(* Logix 5000 project; controller R5_CSS vendor 1 type 14 code 74 rev 19.11; software revision 19.01; part 6 of 20 *)
(* tags used below, declared in another part *)
   AC102A : ANALYTICAL;   // QUENCH WATER CONDUCTIVITY CONTROL
   FC101 : FLOW_CONTROL;   // QUENCH BASIN FLOW TRANSMITTER CONTROL
   FC108 : FLOW_CONTROL;   // QUENCH FEED FLOW TRANSMITTER
   FC140A : FLOW_CONTROL;   // QUENCH TOWER UPPER SPRAY FLOW CONTROL
   FC140B : FLOW_CONTROL;   // QUENCH TOWER LOWER SPRAY FLOW CONTROL
   FC215 : FLOW_CONTROL;   // OVERHEAD CONDENSER CHILLED WATER FLOW CONTROL
   FC365 : FLOW_CONTROL;   // COALESCER PROCESS IMPURITY FLOW CONTROL
   FC370 : FLOW_CONTROL;   // COALESCER MAKE UP WATER FLOW CONTROL
   FC403 : FLOW_CONTROL;   // COALESCER FLOW CONTROLLER FEEDS TCV108
   LCV370_Start : BOOL;
   PID_LC370_Enable : BOOL;
   TMR_FAULT : DINT;
(* MainProgram, continued *)

ROUTINE AT102A_QuenchWaterConductivity   (* ladder *)
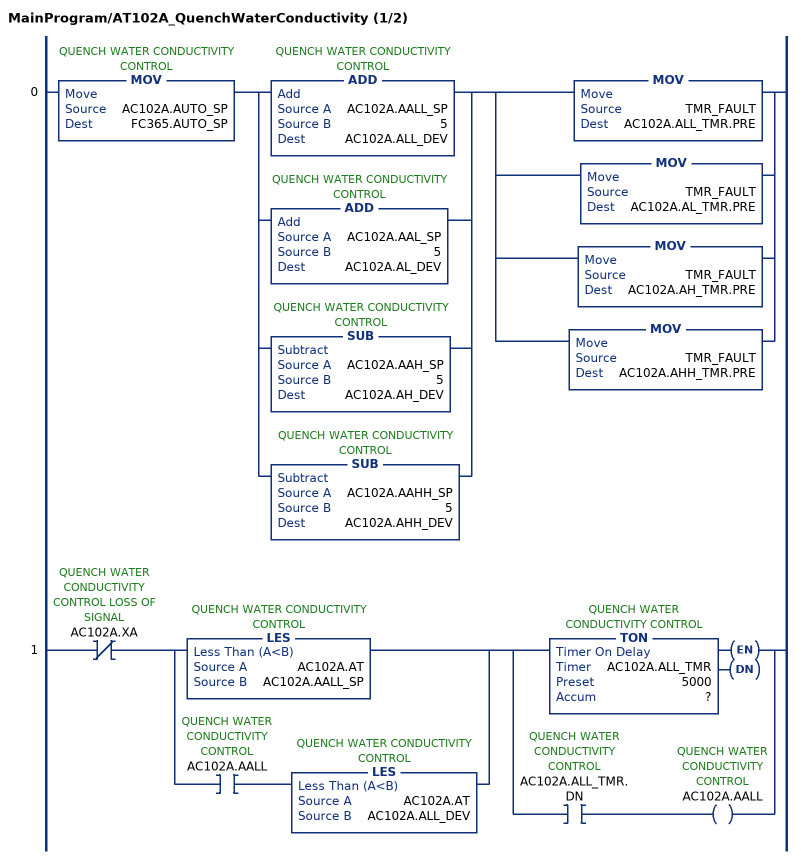
   0: MOV(AC102A.AUTO_SP,FC365.AUTO_SP)[ADD(AC102A.AALL_SP,5,AC102A.ALL_DEV) ,ADD(AC102A.AAL_SP,5,AC102A.AL_DEV) ,SUB(AC102A.AAH_SP,5,AC102A.AH_DEV) ,SUB(AC102A.AAHH_SP,5,AC102A.AHH_DEV) ][MOV(TMR_FAULT,AC102A.ALL_TMR.PRE) ,MOV(TMR_FAULT,AC102A.AL_TMR.PRE) ,MOV(TMR_FAULT,AC102A.AH_TMR.PRE) ,MOV(TMR_FAULT,AC102A.AHH_TMR.PRE) ];
   1: XIO(AC102A.XA)[LES(AC102A.AT,AC102A.AALL_SP) ,XIC(AC102A.AALL) LES(AC102A.AT,AC102A.ALL_DEV) ][TON(AC102A.ALL_TMR,?,?) ,XIC(AC102A.ALL_TMR.DN) OTE(AC102A.AALL) ];
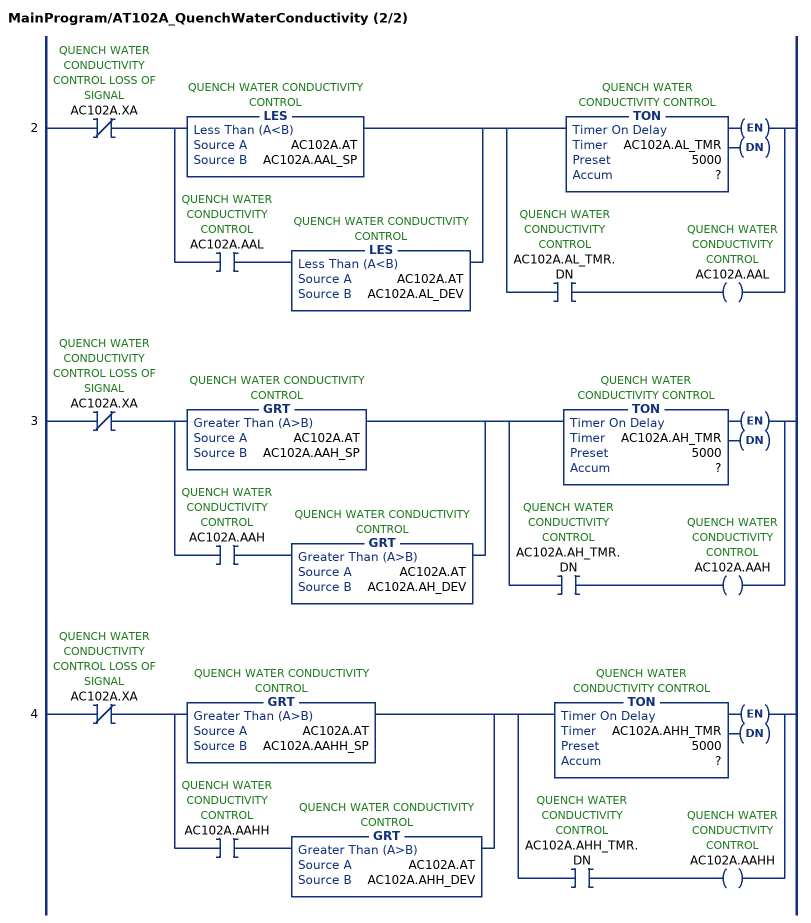
   2: XIO(AC102A.XA)[LES(AC102A.AT,AC102A.AAL_SP) ,XIC(AC102A.AAL) LES(AC102A.AT,AC102A.AL_DEV) ][TON(AC102A.AL_TMR,?,?) ,XIC(AC102A.AL_TMR.DN) OTE(AC102A.AAL) ];
   3: XIO(AC102A.XA)[GRT(AC102A.AT,AC102A.AAH_SP) ,XIC(AC102A.AAH) GRT(AC102A.AT,AC102A.AH_DEV) ][TON(AC102A.AH_TMR,?,?) ,XIC(AC102A.AH_TMR.DN) OTE(AC102A.AAH) ];
   4: XIO(AC102A.XA)[GRT(AC102A.AT,AC102A.AAHH_SP) ,XIC(AC102A.AAHH) GRT(AC102A.AT,AC102A.AHH_DEV) ][TON(AC102A.AHH_TMR,?,?) ,XIC(AC102A.AHH_TMR.DN) OTE(AC102A.AAHH) ];
END_ROUTINE

ROUTINE FC101_BasinFlow   (* ladder *)
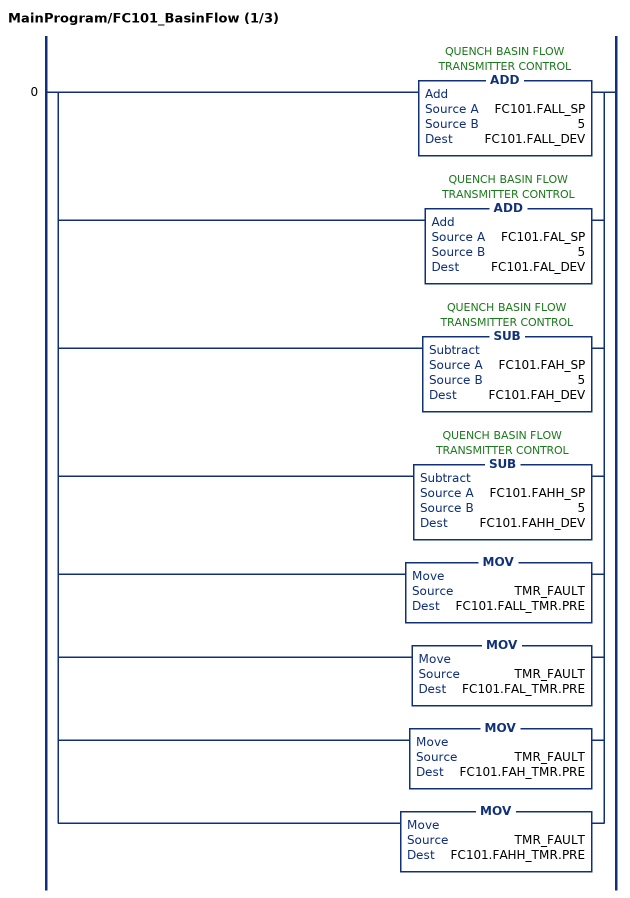
   0: [ADD(FC101.FALL_SP,5,FC101.FALL_DEV) ,ADD(FC101.FAL_SP,5,FC101.FAL_DEV) ,SUB(FC101.FAH_SP,5,FC101.FAH_DEV) ,SUB(FC101.FAHH_SP,5,FC101.FAHH_DEV) ,MOV(TMR_FAULT,FC101.FALL_TMR.PRE) ,MOV(TMR_FAULT,FC101.FAL_TMR.PRE) ,MOV(TMR_FAULT,FC101.FAH_TMR.PRE) ,MOV(TMR_FAULT,FC101.FAHH_TMR.PRE) ];
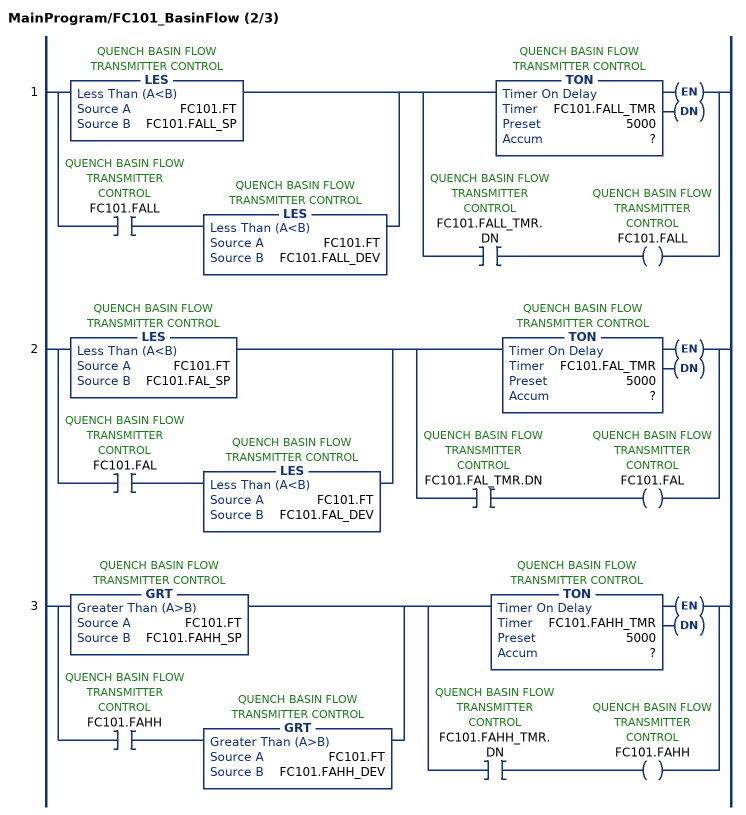
   1: [LES(FC101.FT,FC101.FALL_SP) ,XIC(FC101.FALL) LES(FC101.FT,FC101.FALL_DEV) ][TON(FC101.FALL_TMR,?,?) ,XIC(FC101.FALL_TMR.DN) OTE(FC101.FALL) ];
   2: [LES(FC101.FT,FC101.FAL_SP) ,XIC(FC101.FAL) LES(FC101.FT,FC101.FAL_DEV) ][TON(FC101.FAL_TMR,?,?) ,XIC(FC101.FAL_TMR.DN) OTE(FC101.FAL) ];
   3: [GRT(FC101.FT,FC101.FAHH_SP) ,XIC(FC101.FAHH) GRT(FC101.FT,FC101.FAHH_DEV) ][TON(FC101.FAHH_TMR,?,?) ,XIC(FC101.FAHH_TMR.DN) OTE(FC101.FAHH) ];
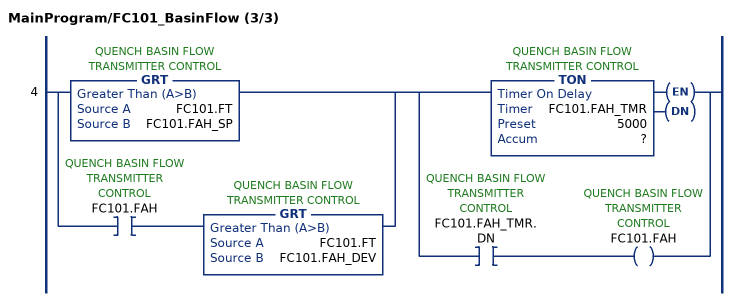
   4: [GRT(FC101.FT,FC101.FAH_SP) ,XIC(FC101.FAH) GRT(FC101.FT,FC101.FAH_DEV) ][TON(FC101.FAH_TMR,?,?) ,XIC(FC101.FAH_TMR.DN) OTE(FC101.FAH) ];
END_ROUTINE

ROUTINE FC108_QuenchTowerFlow   (* ladder *)
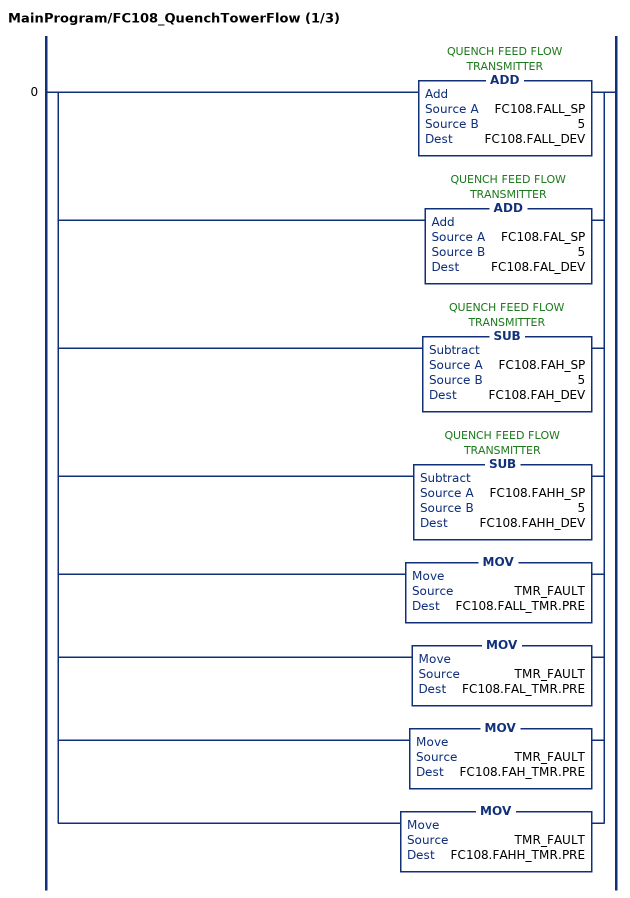
   0: [ADD(FC108.FALL_SP,5,FC108.FALL_DEV) ,ADD(FC108.FAL_SP,5,FC108.FAL_DEV) ,SUB(FC108.FAH_SP,5,FC108.FAH_DEV) ,SUB(FC108.FAHH_SP,5,FC108.FAHH_DEV) ,MOV(TMR_FAULT,FC108.FALL_TMR.PRE) ,MOV(TMR_FAULT,FC108.FAL_TMR.PRE) ,MOV(TMR_FAULT,FC108.FAH_TMR.PRE) ,MOV(TMR_FAULT,FC108.FAHH_TMR.PRE) ];
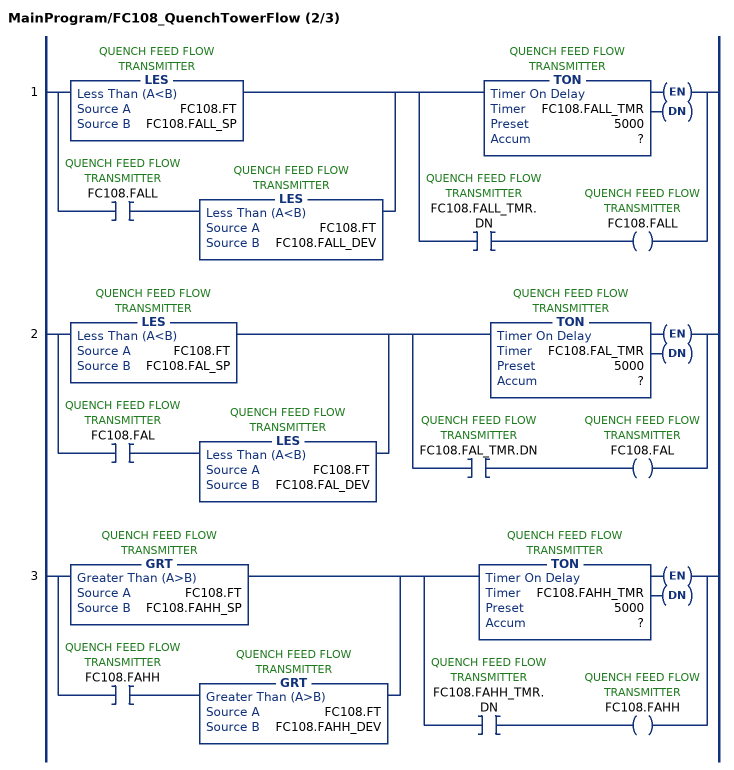
   1: [LES(FC108.FT,FC108.FALL_SP) ,XIC(FC108.FALL) LES(FC108.FT,FC108.FALL_DEV) ][TON(FC108.FALL_TMR,?,?) ,XIC(FC108.FALL_TMR.DN) OTE(FC108.FALL) ];
   2: [LES(FC108.FT,FC108.FAL_SP) ,XIC(FC108.FAL) LES(FC108.FT,FC108.FAL_DEV) ][TON(FC108.FAL_TMR,?,?) ,XIC(FC108.FAL_TMR.DN) OTE(FC108.FAL) ];
   3: [GRT(FC108.FT,FC108.FAHH_SP) ,XIC(FC108.FAHH) GRT(FC108.FT,FC108.FAHH_DEV) ][TON(FC108.FAHH_TMR,?,?) ,XIC(FC108.FAHH_TMR.DN) OTE(FC108.FAHH) ];
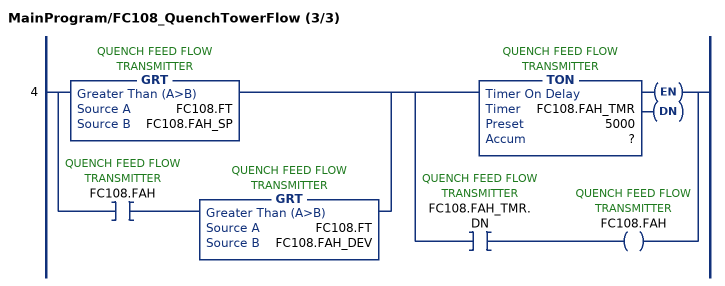
   4: [GRT(FC108.FT,FC108.FAH_SP) ,XIC(FC108.FAH) GRT(FC108.FT,FC108.FAH_DEV) ][TON(FC108.FAH_TMR,?,?) ,XIC(FC108.FAH_TMR.DN) OTE(FC108.FAH) ];
END_ROUTINE

ROUTINE FC140A_QuenchWaterUpperSprayFlow   (* ladder *)
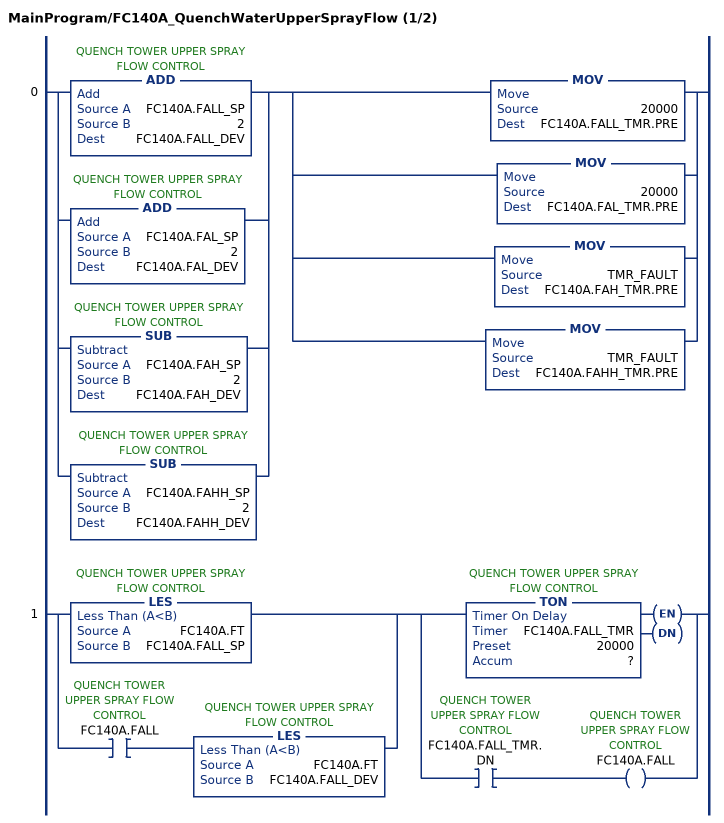
   0: [ADD(FC140A.FALL_SP,2,FC140A.FALL_DEV) ,ADD(FC140A.FAL_SP,2,FC140A.FAL_DEV) ,SUB(FC140A.FAH_SP,2,FC140A.FAH_DEV) ,SUB(FC140A.FAHH_SP,2,FC140A.FAHH_DEV) ][MOV(20000,FC140A.FALL_TMR.PRE) ,MOV(20000,FC140A.FAL_TMR.PRE) ,MOV(TMR_FAULT,FC140A.FAH_TMR.PRE) ,MOV(TMR_FAULT,FC140A.FAHH_TMR.PRE) ];
   1: [LES(FC140A.FT,FC140A.FALL_SP) ,XIC(FC140A.FALL) LES(FC140A.FT,FC140A.FALL_DEV) ][TON(FC140A.FALL_TMR,?,?) ,XIC(FC140A.FALL_TMR.DN) OTE(FC140A.FALL) ];
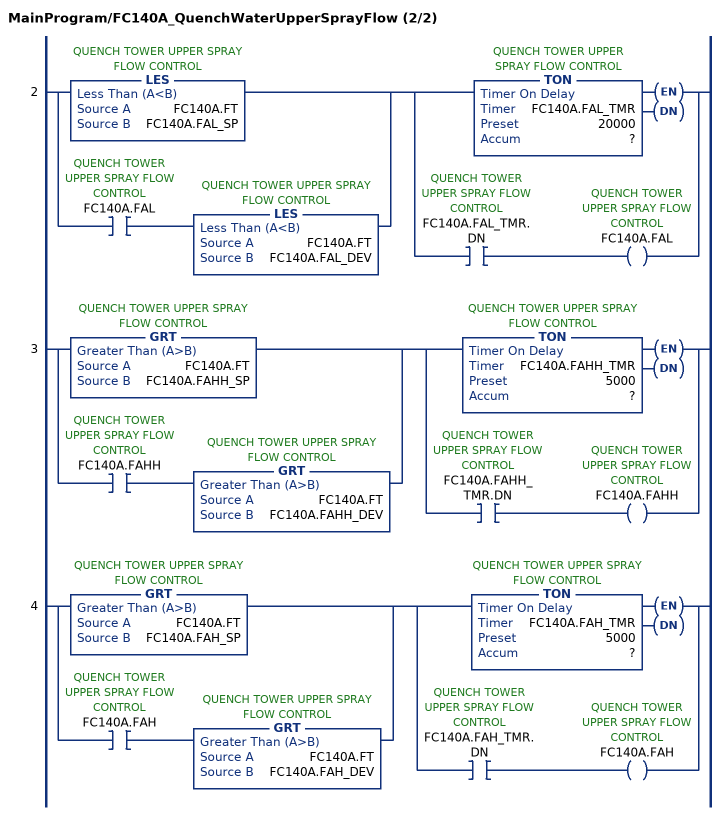
   2: [LES(FC140A.FT,FC140A.FAL_SP) ,XIC(FC140A.FAL) LES(FC140A.FT,FC140A.FAL_DEV) ][TON(FC140A.FAL_TMR,?,?) ,XIC(FC140A.FAL_TMR.DN) OTE(FC140A.FAL) ];
   3: [GRT(FC140A.FT,FC140A.FAHH_SP) ,XIC(FC140A.FAHH) GRT(FC140A.FT,FC140A.FAHH_DEV) ][TON(FC140A.FAHH_TMR,?,?) ,XIC(FC140A.FAHH_TMR.DN) OTE(FC140A.FAHH) ];
   4: [GRT(FC140A.FT,FC140A.FAH_SP) ,XIC(FC140A.FAH) GRT(FC140A.FT,FC140A.FAH_DEV) ][TON(FC140A.FAH_TMR,?,?) ,XIC(FC140A.FAH_TMR.DN) OTE(FC140A.FAH) ];
END_ROUTINE

ROUTINE FC140B_QuenchWaterLowerSprayFlow   (* ladder *)
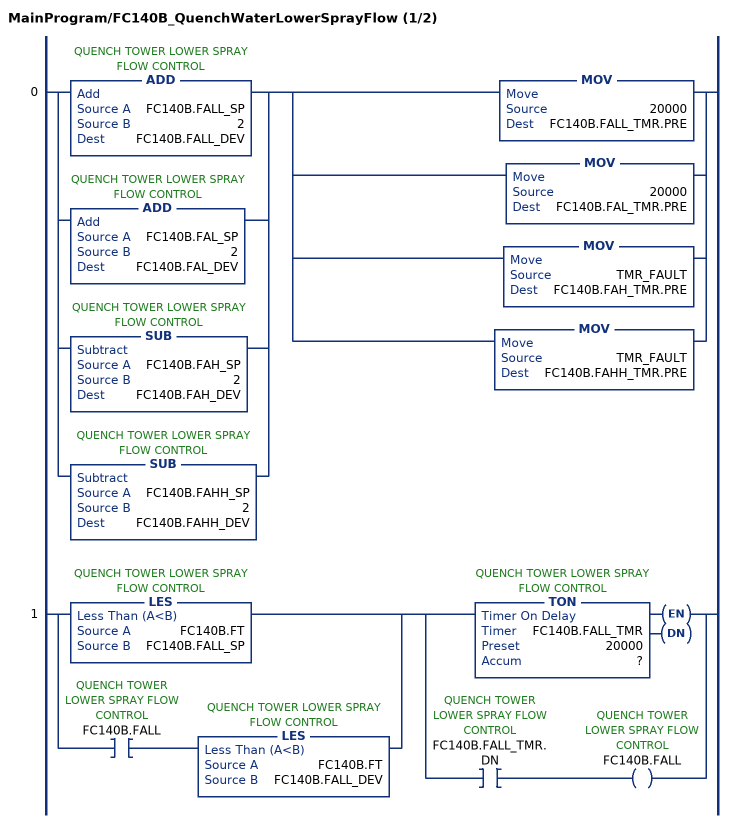
   0: [ADD(FC140B.FALL_SP,2,FC140B.FALL_DEV) ,ADD(FC140B.FAL_SP,2,FC140B.FAL_DEV) ,SUB(FC140B.FAH_SP,2,FC140B.FAH_DEV) ,SUB(FC140B.FAHH_SP,2,FC140B.FAHH_DEV) ][MOV(20000,FC140B.FALL_TMR.PRE) ,MOV(20000,FC140B.FAL_TMR.PRE) ,MOV(TMR_FAULT,FC140B.FAH_TMR.PRE) ,MOV(TMR_FAULT,FC140B.FAHH_TMR.PRE) ];
   1: [LES(FC140B.FT,FC140B.FALL_SP) ,XIC(FC140B.FALL) LES(FC140B.FT,FC140B.FALL_DEV) ][TON(FC140B.FALL_TMR,?,?) ,XIC(FC140B.FALL_TMR.DN) OTE(FC140B.FALL) ];
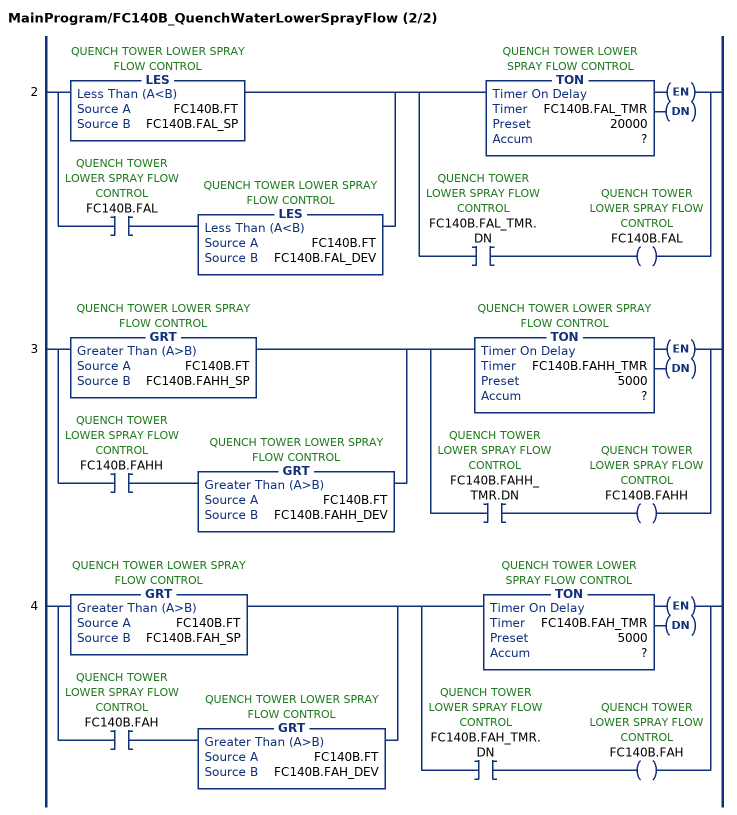
   2: [LES(FC140B.FT,FC140B.FAL_SP) ,XIC(FC140B.FAL) LES(FC140B.FT,FC140B.FAL_DEV) ][TON(FC140B.FAL_TMR,?,?) ,XIC(FC140B.FAL_TMR.DN) OTE(FC140B.FAL) ];
   3: [GRT(FC140B.FT,FC140B.FAHH_SP) ,XIC(FC140B.FAHH) GRT(FC140B.FT,FC140B.FAHH_DEV) ][TON(FC140B.FAHH_TMR,?,?) ,XIC(FC140B.FAHH_TMR.DN) OTE(FC140B.FAHH) ];
   4: [GRT(FC140B.FT,FC140B.FAH_SP) ,XIC(FC140B.FAH) GRT(FC140B.FT,FC140B.FAH_DEV) ][TON(FC140B.FAH_TMR,?,?) ,XIC(FC140B.FAH_TMR.DN) OTE(FC140B.FAH) ];
END_ROUTINE

ROUTINE FC215_OverheadCondChillWaterFlow   (* ladder *)
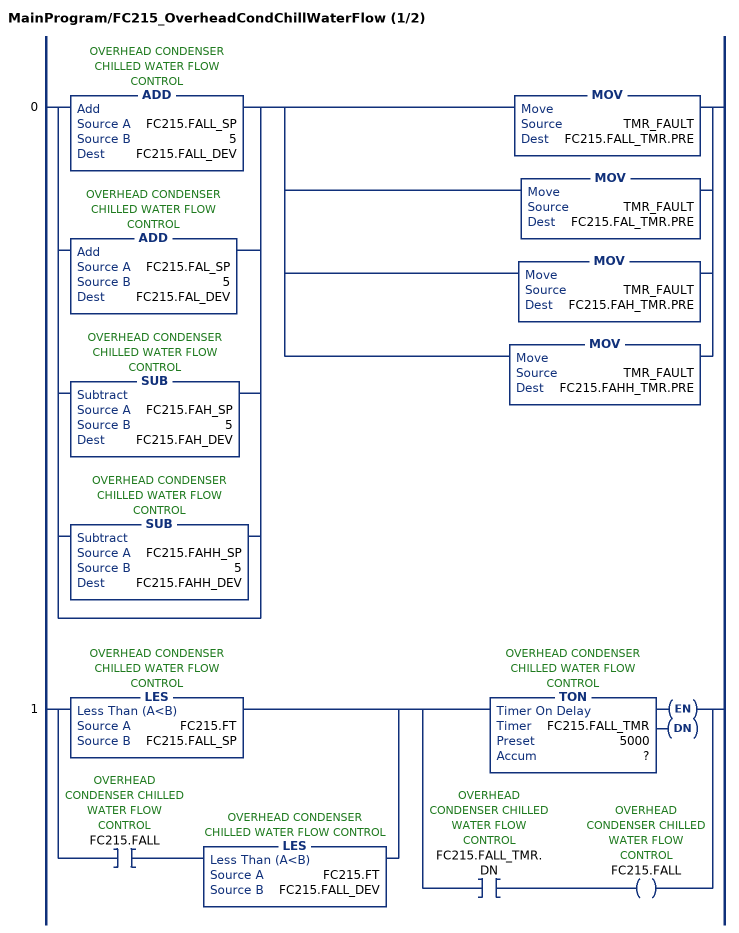
   0: [ADD(FC215.FALL_SP,5,FC215.FALL_DEV) ,ADD(FC215.FAL_SP,5,FC215.FAL_DEV) ,SUB(FC215.FAH_SP,5,FC215.FAH_DEV) ,SUB(FC215.FAHH_SP,5,FC215.FAHH_DEV) ,][MOV(TMR_FAULT,FC215.FALL_TMR.PRE) ,MOV(TMR_FAULT,FC215.FAL_TMR.PRE) ,MOV(TMR_FAULT,FC215.FAH_TMR.PRE) ,MOV(TMR_FAULT,FC215.FAHH_TMR.PRE) ];
   1: [LES(FC215.FT,FC215.FALL_SP) ,XIC(FC215.FALL) LES(FC215.FT,FC215.FALL_DEV) ][TON(FC215.FALL_TMR,?,?) ,XIC(FC215.FALL_TMR.DN) OTE(FC215.FALL) ];
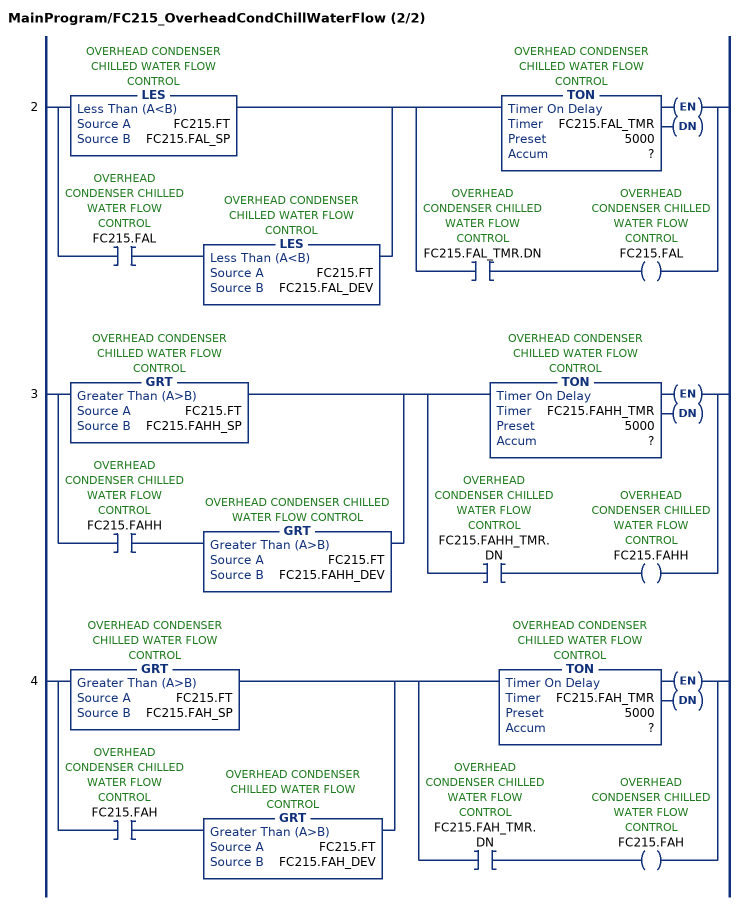
   2: [LES(FC215.FT,FC215.FAL_SP) ,XIC(FC215.FAL) LES(FC215.FT,FC215.FAL_DEV) ][TON(FC215.FAL_TMR,?,?) ,XIC(FC215.FAL_TMR.DN) OTE(FC215.FAL) ];
   3: [GRT(FC215.FT,FC215.FAHH_SP) ,XIC(FC215.FAHH) GRT(FC215.FT,FC215.FAHH_DEV) ][TON(FC215.FAHH_TMR,?,?) ,XIC(FC215.FAHH_TMR.DN) OTE(FC215.FAHH) ];
   4: [GRT(FC215.FT,FC215.FAH_SP) ,XIC(FC215.FAH) GRT(FC215.FT,FC215.FAH_DEV) ][TON(FC215.FAH_TMR,?,?) ,XIC(FC215.FAH_TMR.DN) OTE(FC215.FAH) ];
END_ROUTINE

ROUTINE FC370_WaterMakeupFlow   (* ladder *)
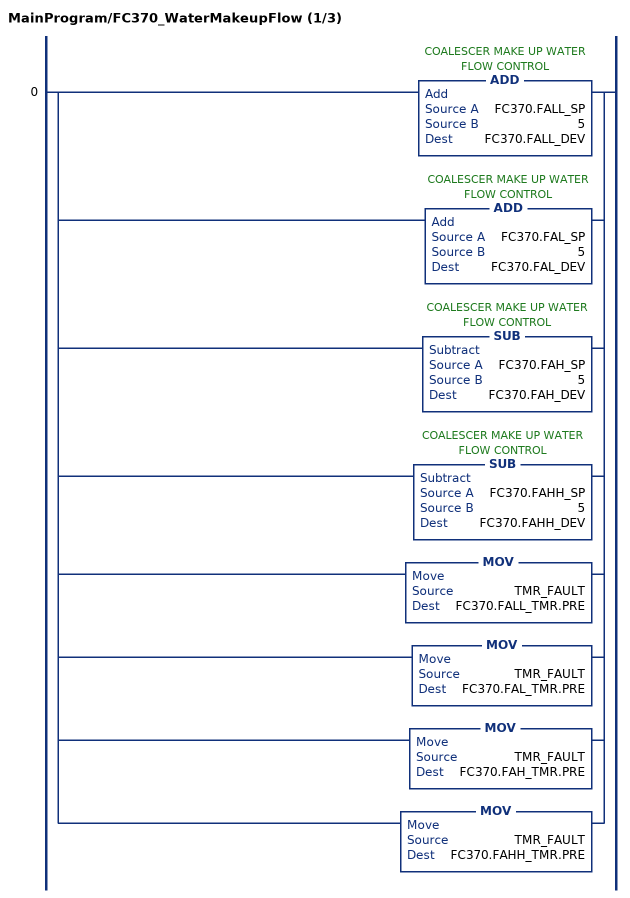
   0: [ADD(FC370.FALL_SP,5,FC370.FALL_DEV) ,ADD(FC370.FAL_SP,5,FC370.FAL_DEV) ,SUB(FC370.FAH_SP,5,FC370.FAH_DEV) ,SUB(FC370.FAHH_SP,5,FC370.FAHH_DEV) ,MOV(TMR_FAULT,FC370.FALL_TMR.PRE) ,MOV(TMR_FAULT,FC370.FAL_TMR.PRE) ,MOV(TMR_FAULT,FC370.FAH_TMR.PRE) ,MOV(TMR_FAULT,FC370.FAHH_TMR.PRE) ];
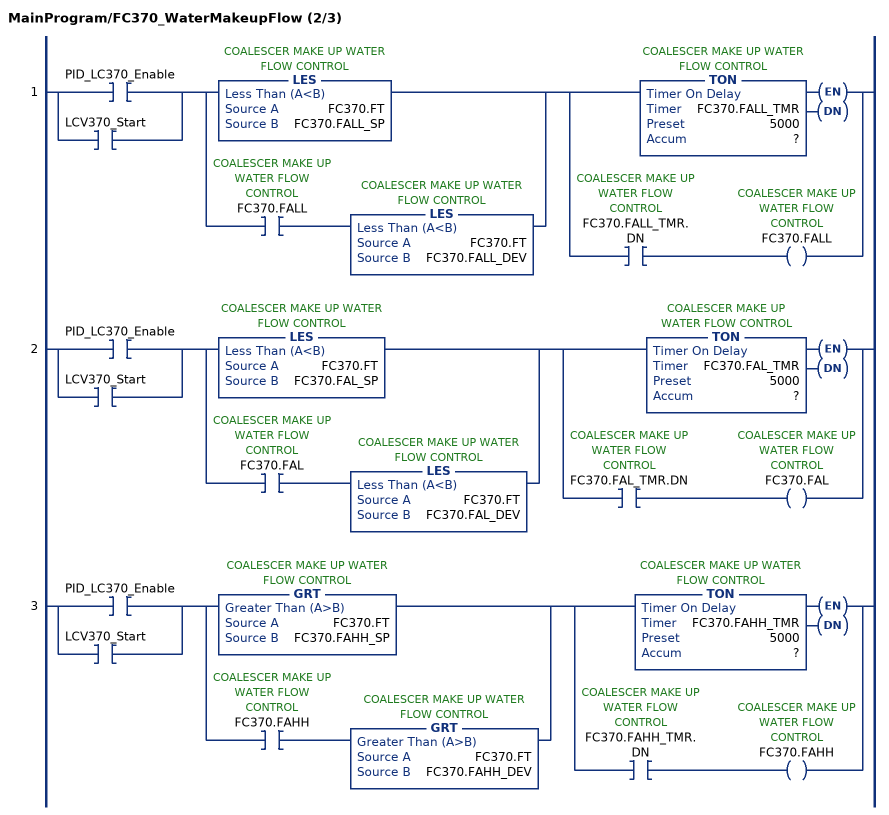
   1: [XIC(PID_LC370_Enable) ,XIC(LCV370_Start) ][LES(FC370.FT,FC370.FALL_SP) ,XIC(FC370.FALL) LES(FC370.FT,FC370.FALL_DEV) ][TON(FC370.FALL_TMR,?,?) ,XIC(FC370.FALL_TMR.DN) OTE(FC370.FALL) ];
   2: [XIC(PID_LC370_Enable) ,XIC(LCV370_Start) ][LES(FC370.FT,FC370.FAL_SP) ,XIC(FC370.FAL) LES(FC370.FT,FC370.FAL_DEV) ][TON(FC370.FAL_TMR,?,?) ,XIC(FC370.FAL_TMR.DN) OTE(FC370.FAL) ];
   3: [XIC(PID_LC370_Enable) ,XIC(LCV370_Start) ][GRT(FC370.FT,FC370.FAHH_SP) ,XIC(FC370.FAHH) GRT(FC370.FT,FC370.FAHH_DEV) ][TON(FC370.FAHH_TMR,?,?) ,XIC(FC370.FAHH_TMR.DN) OTE(FC370.FAHH) ];
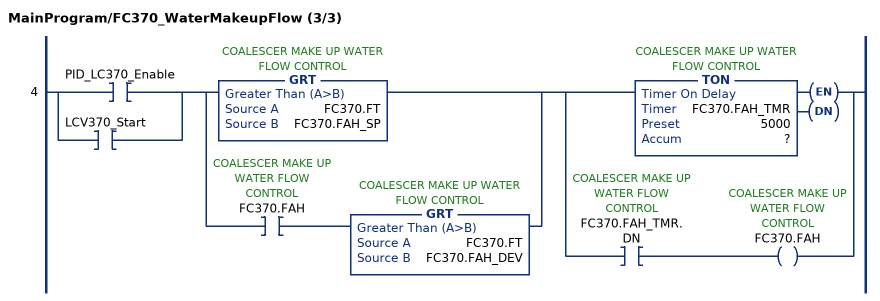
   4: [XIC(PID_LC370_Enable) ,XIC(LCV370_Start) ][GRT(FC370.FT,FC370.FAH_SP) ,XIC(FC370.FAH) GRT(FC370.FT,FC370.FAH_DEV) ][TON(FC370.FAH_TMR,?,?) ,XIC(FC370.FAH_TMR.DN) OTE(FC370.FAH) ];
END_ROUTINE

ROUTINE FC403_QuenchWaterTotalFlow   (* ladder *)
// COALESCER FLOW CONTROL
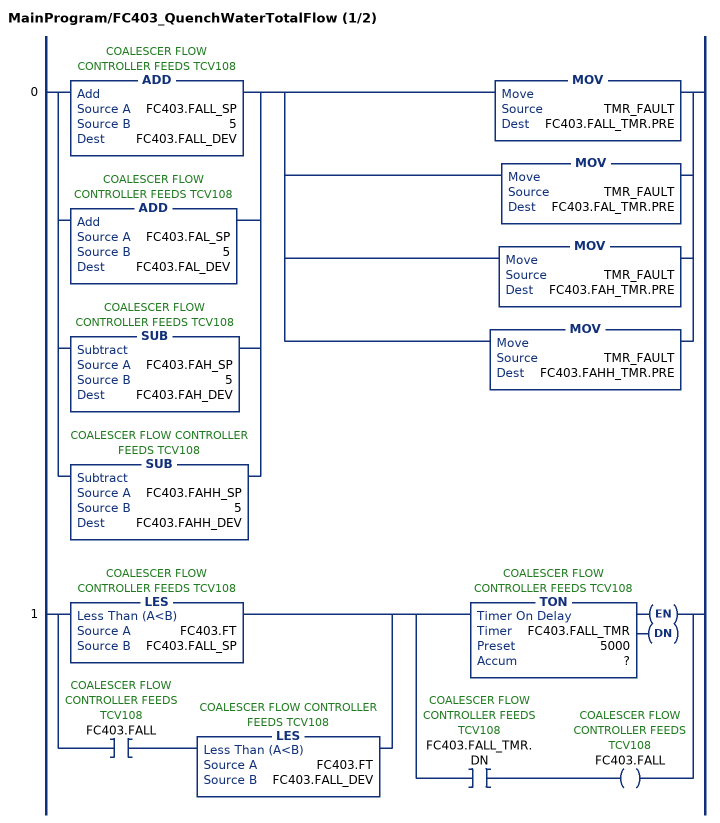
   0: [ADD(FC403.FALL_SP,5,FC403.FALL_DEV) ,ADD(FC403.FAL_SP,5,FC403.FAL_DEV) ,SUB(FC403.FAH_SP,5,FC403.FAH_DEV) ,SUB(FC403.FAHH_SP,5,FC403.FAHH_DEV) ][MOV(TMR_FAULT,FC403.FALL_TMR.PRE) ,MOV(TMR_FAULT,FC403.FAL_TMR.PRE) ,MOV(TMR_FAULT,FC403.FAH_TMR.PRE) ,MOV(TMR_FAULT,FC403.FAHH_TMR.PRE) ];
   1: [LES(FC403.FT,FC403.FALL_SP) ,XIC(FC403.FALL) LES(FC403.FT,FC403.FALL_DEV) ][TON(FC403.FALL_TMR,?,?) ,XIC(FC403.FALL_TMR.DN) OTE(FC403.FALL) ];
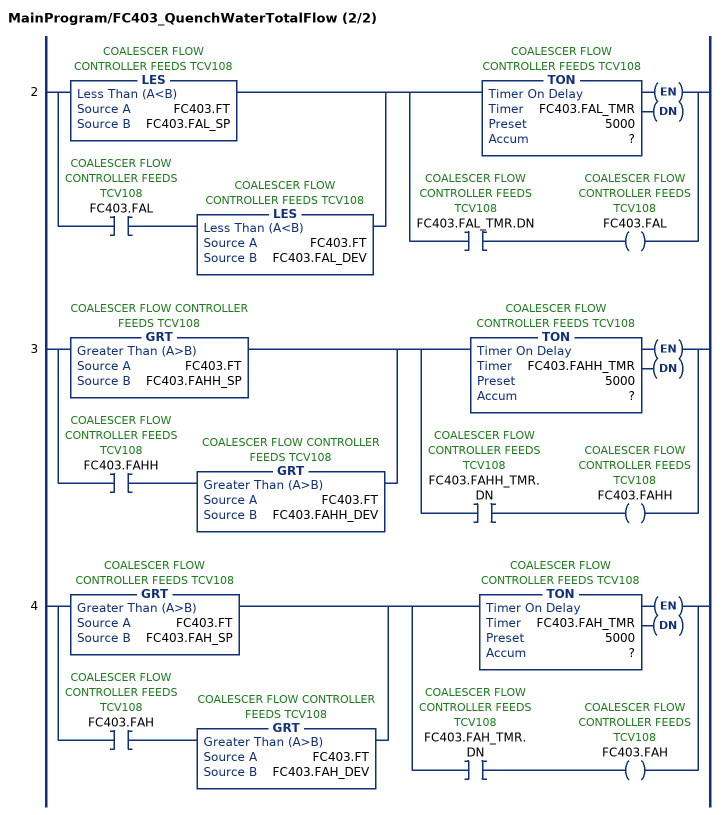
   2: [LES(FC403.FT,FC403.FAL_SP) ,XIC(FC403.FAL) LES(FC403.FT,FC403.FAL_DEV) ][TON(FC403.FAL_TMR,?,?) ,XIC(FC403.FAL_TMR.DN) OTE(FC403.FAL) ];
   3: [GRT(FC403.FT,FC403.FAHH_SP) ,XIC(FC403.FAHH) GRT(FC403.FT,FC403.FAHH_DEV) ][TON(FC403.FAHH_TMR,?,?) ,XIC(FC403.FAHH_TMR.DN) OTE(FC403.FAHH) ];
   4: [GRT(FC403.FT,FC403.FAH_SP) ,XIC(FC403.FAH) GRT(FC403.FT,FC403.FAH_DEV) ][TON(FC403.FAH_TMR,?,?) ,XIC(FC403.FAH_TMR.DN) OTE(FC403.FAH) ];
END_ROUTINE
